FUNCTION_BLOCK FB_ListObjectTests EXTENDS 
VAR_INPUT
END_VAR
VAR_OUTPUT
	fbTestsuite:			FB_Testsuite;
END_VAR
VAR
	fbList:					Tc3_Component.FB_ListObject;
	fbObject:				Tc3_Component.FB_Object;
	iObject:				Tc3_Component.I_Object:= fbObject;
END_VAR

fbTestsuite.P_Property.M_Add('object', 'FB_ListObject');
fbTestsuite.P_Property.M_Add('name', 'Peter Zerlauth');

fbTestsuite();

CASE fbTestsuite.P_Testcase OF
	
	E_Testcase.Start:
		fbTestsuite.P_Assert.M_Equals_DINT(fbList.P_Length, 0, 'P_Length');
		fbTestsuite.M_Testcase('FB_ListObject', T#2S, 'fbList.P_Length', '', 10);	
		
	10:
		fbTestsuite.P_Assert.M_Equals_BOOL(fbList.M_Add(fbObject), TRUE, 'M_Add(fbObject)');
		fbTestsuite.M_Testcase('FB_ListObject', T#2S, 'fbList.M_Add(fbObject)', '', 20);
		
	20:
		fbTestsuite.P_Assert.M_Equals_DINT(fbList.P_Length, 1, 'P_Length');
		fbTestsuite.M_Testcase('FB_ListObject', T#2S, 'fbList.P_Length', '', 30);		
		
	30:
		fbTestsuite.P_Assert.M_Equals_DINT(fbList.M_Find(fbObject), 0, 'M_Find');
		fbTestsuite.M_Testcase('FB_ListObject', T#2S, 'fbList.M_Find(fbObject)', '', 40);
		
	40:

		fbTestsuite.P_Assert.M_Equals_BOOL(TRUE, __QUERYINTERFACE(fbList.M_Index(0), iObject), 'M_Index');
		fbTestsuite.M_Testcase('FB_ListObject', T#2S, 'fbList.M_Index(1)', '', 50);
		
	50:
		fbTestsuite.P_Assert.M_Equals_BOOL(fbList.M_Remove(fbObject), TRUE, 'M_Remove');
		fbTestsuite.M_Testcase('FB_ListObject', T#2S, 'fbList.M_Remove(fbObject', '', 60);		

	60:
		fbTestsuite.P_Assert.M_Equals_DINT(fbList.P_Length, 0, 'P_Length');
		fbTestsuite.M_Testcase('FB_ListObject', T#2S, 'fbList.P_Length', '', 70);
		
	70:
		fbTestsuite.P_Assert.M_Equals_BOOL(fbList.M_Add(fbObject), TRUE, 'M_Add(fbObject)');
		fbTestsuite.M_Testcase('FB_ListObject', T#2S, 'fbList.M_Add(fbObject)', '', 80);

	80:
		fbTestsuite.P_Assert.M_Equals_DINT(fbList.P_Length, 1, 'P_Length');
		fbTestsuite.M_Testcase('FB_ListObject', T#2S, 'fbList.P_Length', '', 90);
		
	90:
		fbTestsuite.P_Assert.M_Equals_BOOL(fbList.M_Clear(), TRUE, 'M_Clear()');
		fbTestsuite.M_Testcase('FB_ListObject', T#2S, 'fbList.M_Clear()', '', 100);		
	
	100:
		fbTestsuite.P_Assert.M_Equals_DINT(fbList.P_Length, 0, 'P_Length');
		fbTestsuite.M_Testcase('FB_ListObject', T#2S, 'fbList.P_Length', '', E_Testcase.Done);
		
	E_Testcase.Done:
	
END_CASE

END_FUNCTION_BLOCK

(* stored: Version 1.1.0.1
   POU FB_ListObjectTests: Id {fa7d1354-c4bf-0027-35b9-9e4297f35a74}, SpecialFunc None *)
